(* PLC project 未命名, 未知 未命名 1 *)
(* stored: creationDateTime 2021-06-18T11:02:46, modificationDateTime 2021-06-18T15:59:58 *)

PROGRAM helloword
  VAR
    PB1 AT %IX0.0 : BOOL;
    PB2 AT %IX0.1 : BOOL;
    LED AT %QX0.0 : BOOL;
  END_VAR

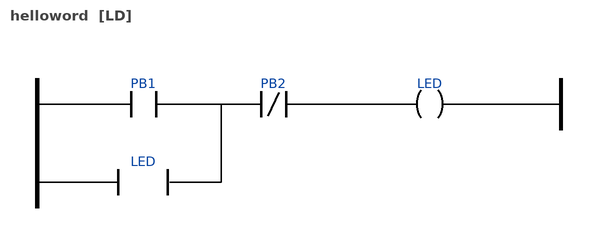
(* LD diagram, written out as Structured Text *)
LED := (PB1 OR LED) AND NOT PB2;
END_PROGRAM

CONFIGURATION Config0
  RESOURCE Res0 ON PLC
    TASK task0(INTERVAL := T#20ms, PRIORITY := 0);
    PROGRAM instance0 WITH task0 : helloword;
  END_RESOURCE
END_CONFIGURATION
